REGION Network 24: Position Teaching (No 29~32)
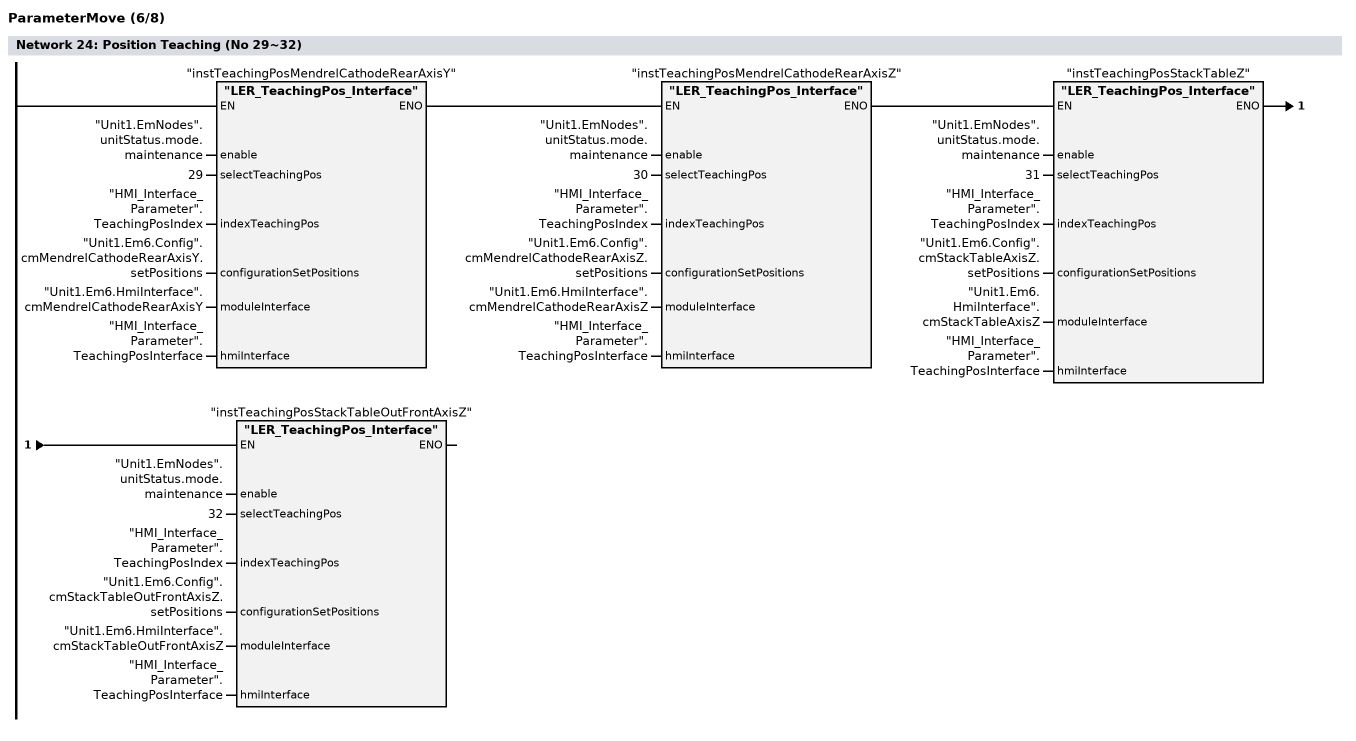
   RUNG wire#powerrail
      "instTeachingPosMendrelCathodeRearAxisY"(enable := "Unit1.EmNodes".unitStatus.mode.maintenance, selectTeachingPos := 29, indexTeachingPos := "HMI_Interface_Parameter".TeachingPosIndex, configurationSetPositions := "Unit1.Em6.Config".cmMendrelCathodeRearAxisY.setPositions, moduleInterface := "Unit1.Em6.HmiInterface".cmMendrelCathodeRearAxisY, hmiInterface := "HMI_Interface_Parameter".TeachingPosInterface)
      "instTeachingPosMendrelCathodeRearAxisZ"(enable := "Unit1.EmNodes".unitStatus.mode.maintenance, selectTeachingPos := 30, indexTeachingPos := "HMI_Interface_Parameter".TeachingPosIndex, configurationSetPositions := "Unit1.Em6.Config".cmMendrelCathodeRearAxisZ.setPositions, moduleInterface := "Unit1.Em6.HmiInterface".cmMendrelCathodeRearAxisZ, hmiInterface := "HMI_Interface_Parameter".TeachingPosInterface)
      "instTeachingPosStackTableZ"(enable := "Unit1.EmNodes".unitStatus.mode.maintenance, selectTeachingPos := 31, indexTeachingPos := "HMI_Interface_Parameter".TeachingPosIndex, configurationSetPositions := "Unit1.Em6.Config".cmStackTableAxisZ.setPositions, moduleInterface := "Unit1.Em6.HmiInterface".cmStackTableAxisZ, hmiInterface := "HMI_Interface_Parameter".TeachingPosInterface)
      "instTeachingPosStackTableOutFrontAxisZ"(enable := "Unit1.EmNodes".unitStatus.mode.maintenance, selectTeachingPos := 32, indexTeachingPos := "HMI_Interface_Parameter".TeachingPosIndex, configurationSetPositions := "Unit1.Em6.Config".cmStackTableOutFrontAxisZ.setPositions, moduleInterface := "Unit1.Em6.HmiInterface".cmStackTableOutFrontAxisZ, hmiInterface := "HMI_Interface_Parameter".TeachingPosInterface)
   END_RUNG
   // the same network as SCL:
   "instTeachingPosMendrelCathodeRearAxisY"(enable := "Unit1.EmNodes".unitStatus.mode.maintenance,   // "LER_TeachingPos_Interface"
                           selectTeachingPos := 29,
                           indexTeachingPos := "HMI_Interface_Parameter".TeachingPosIndex,
                           configurationSetPositions := "Unit1.Em6.Config".cmMendrelCathodeRearAxisY.setPositions,
                           moduleInterface := "Unit1.Em6.HmiInterface".cmMendrelCathodeRearAxisY,
                           hmiInterface := "HMI_Interface_Parameter".TeachingPosInterface,
                           ENO => #_w1);
   "instTeachingPosMendrelCathodeRearAxisZ"(EN := #_w1,   // "LER_TeachingPos_Interface"
                           enable := "Unit1.EmNodes".unitStatus.mode.maintenance,
                           selectTeachingPos := 30,
                           indexTeachingPos := "HMI_Interface_Parameter".TeachingPosIndex,
                           configurationSetPositions := "Unit1.Em6.Config".cmMendrelCathodeRearAxisZ.setPositions,
                           moduleInterface := "Unit1.Em6.HmiInterface".cmMendrelCathodeRearAxisZ,
                           hmiInterface := "HMI_Interface_Parameter".TeachingPosInterface,
                           ENO => #_w2);
   "instTeachingPosStackTableZ"(EN := #_w2,   // "LER_TeachingPos_Interface"
                           enable := "Unit1.EmNodes".unitStatus.mode.maintenance,
                           selectTeachingPos := 31,
                           indexTeachingPos := "HMI_Interface_Parameter".TeachingPosIndex,
                           configurationSetPositions := "Unit1.Em6.Config".cmStackTableAxisZ.setPositions,
                           moduleInterface := "Unit1.Em6.HmiInterface".cmStackTableAxisZ,
                           hmiInterface := "HMI_Interface_Parameter".TeachingPosInterface,
                           ENO => #_w3);
   IF #_w3 THEN
       "instTeachingPosStackTableOutFrontAxisZ"(enable := "Unit1.EmNodes".unitStatus.mode.maintenance,   // "LER_TeachingPos_Interface"
                               selectTeachingPos := 32,
                               indexTeachingPos := "HMI_Interface_Parameter".TeachingPosIndex,
                               configurationSetPositions := "Unit1.Em6.Config".cmStackTableOutFrontAxisZ.setPositions,
                               moduleInterface := "Unit1.Em6.HmiInterface".cmStackTableOutFrontAxisZ,
                               hmiInterface := "HMI_Interface_Parameter".TeachingPosInterface);
   END_IF;
END_REGION

REGION Network 25: Position Teaching (No 33~36)
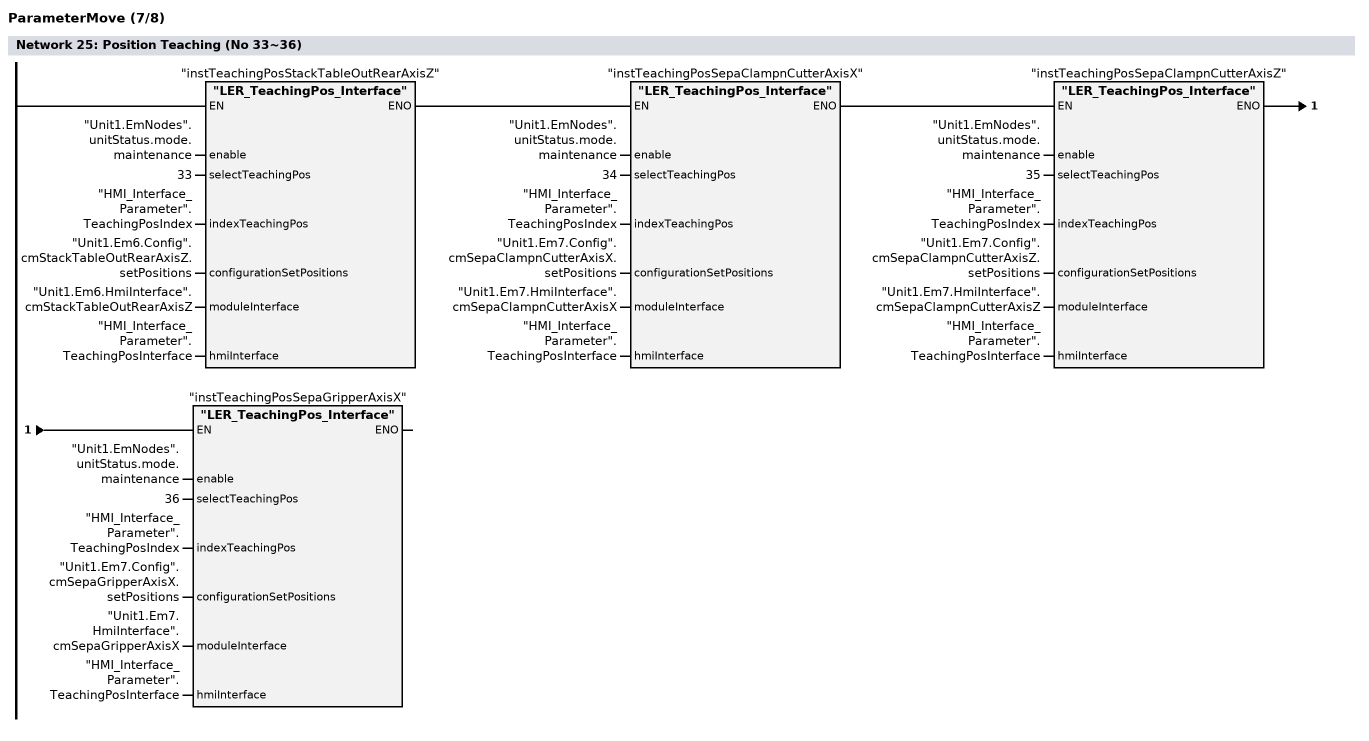
   RUNG wire#powerrail
      "instTeachingPosStackTableOutRearAxisZ"(enable := "Unit1.EmNodes".unitStatus.mode.maintenance, selectTeachingPos := 33, indexTeachingPos := "HMI_Interface_Parameter".TeachingPosIndex, configurationSetPositions := "Unit1.Em6.Config".cmStackTableOutRearAxisZ.setPositions, moduleInterface := "Unit1.Em6.HmiInterface".cmStackTableOutRearAxisZ, hmiInterface := "HMI_Interface_Parameter".TeachingPosInterface)
      "instTeachingPosSepaClampnCutterAxisX"(enable := "Unit1.EmNodes".unitStatus.mode.maintenance, selectTeachingPos := 34, indexTeachingPos := "HMI_Interface_Parameter".TeachingPosIndex, configurationSetPositions := "Unit1.Em7.Config".cmSepaClampnCutterAxisX.setPositions, moduleInterface := "Unit1.Em7.HmiInterface".cmSepaClampnCutterAxisX, hmiInterface := "HMI_Interface_Parameter".TeachingPosInterface)
      "instTeachingPosSepaClampnCutterAxisZ"(enable := "Unit1.EmNodes".unitStatus.mode.maintenance, selectTeachingPos := 35, indexTeachingPos := "HMI_Interface_Parameter".TeachingPosIndex, configurationSetPositions := "Unit1.Em7.Config".cmSepaClampnCutterAxisZ.setPositions, moduleInterface := "Unit1.Em7.HmiInterface".cmSepaClampnCutterAxisZ, hmiInterface := "HMI_Interface_Parameter".TeachingPosInterface)
      "instTeachingPosSepaGripperAxisX"(enable := "Unit1.EmNodes".unitStatus.mode.maintenance, selectTeachingPos := 36, indexTeachingPos := "HMI_Interface_Parameter".TeachingPosIndex, configurationSetPositions := "Unit1.Em7.Config".cmSepaGripperAxisX.setPositions, moduleInterface := "Unit1.Em7.HmiInterface".cmSepaGripperAxisX, hmiInterface := "HMI_Interface_Parameter".TeachingPosInterface)
   END_RUNG
   // the same network as SCL:
   "instTeachingPosStackTableOutRearAxisZ"(enable := "Unit1.EmNodes".unitStatus.mode.maintenance,   // "LER_TeachingPos_Interface"
                           selectTeachingPos := 33,
                           indexTeachingPos := "HMI_Interface_Parameter".TeachingPosIndex,
                           configurationSetPositions := "Unit1.Em6.Config".cmStackTableOutRearAxisZ.setPositions,
                           moduleInterface := "Unit1.Em6.HmiInterface".cmStackTableOutRearAxisZ,
                           hmiInterface := "HMI_Interface_Parameter".TeachingPosInterface,
                           ENO => #_w1);
   "instTeachingPosSepaClampnCutterAxisX"(EN := #_w1,   // "LER_TeachingPos_Interface"
                           enable := "Unit1.EmNodes".unitStatus.mode.maintenance,
                           selectTeachingPos := 34,
                           indexTeachingPos := "HMI_Interface_Parameter".TeachingPosIndex,
                           configurationSetPositions := "Unit1.Em7.Config".cmSepaClampnCutterAxisX.setPositions,
                           moduleInterface := "Unit1.Em7.HmiInterface".cmSepaClampnCutterAxisX,
                           hmiInterface := "HMI_Interface_Parameter".TeachingPosInterface,
                           ENO => #_w2);
   "instTeachingPosSepaClampnCutterAxisZ"(EN := #_w2,   // "LER_TeachingPos_Interface"
                           enable := "Unit1.EmNodes".unitStatus.mode.maintenance,
                           selectTeachingPos := 35,
                           indexTeachingPos := "HMI_Interface_Parameter".TeachingPosIndex,
                           configurationSetPositions := "Unit1.Em7.Config".cmSepaClampnCutterAxisZ.setPositions,
                           moduleInterface := "Unit1.Em7.HmiInterface".cmSepaClampnCutterAxisZ,
                           hmiInterface := "HMI_Interface_Parameter".TeachingPosInterface,
                           ENO => #_w3);
   IF #_w3 THEN
       "instTeachingPosSepaGripperAxisX"(enable := "Unit1.EmNodes".unitStatus.mode.maintenance,   // "LER_TeachingPos_Interface"
                               selectTeachingPos := 36,
                               indexTeachingPos := "HMI_Interface_Parameter".TeachingPosIndex,
                               configurationSetPositions := "Unit1.Em7.Config".cmSepaGripperAxisX.setPositions,
                               moduleInterface := "Unit1.Em7.HmiInterface".cmSepaGripperAxisX,
                               hmiInterface := "HMI_Interface_Parameter".TeachingPosInterface);
   END_IF;
END_REGION

REGION Network 26: Position Teaching (No 37~40)
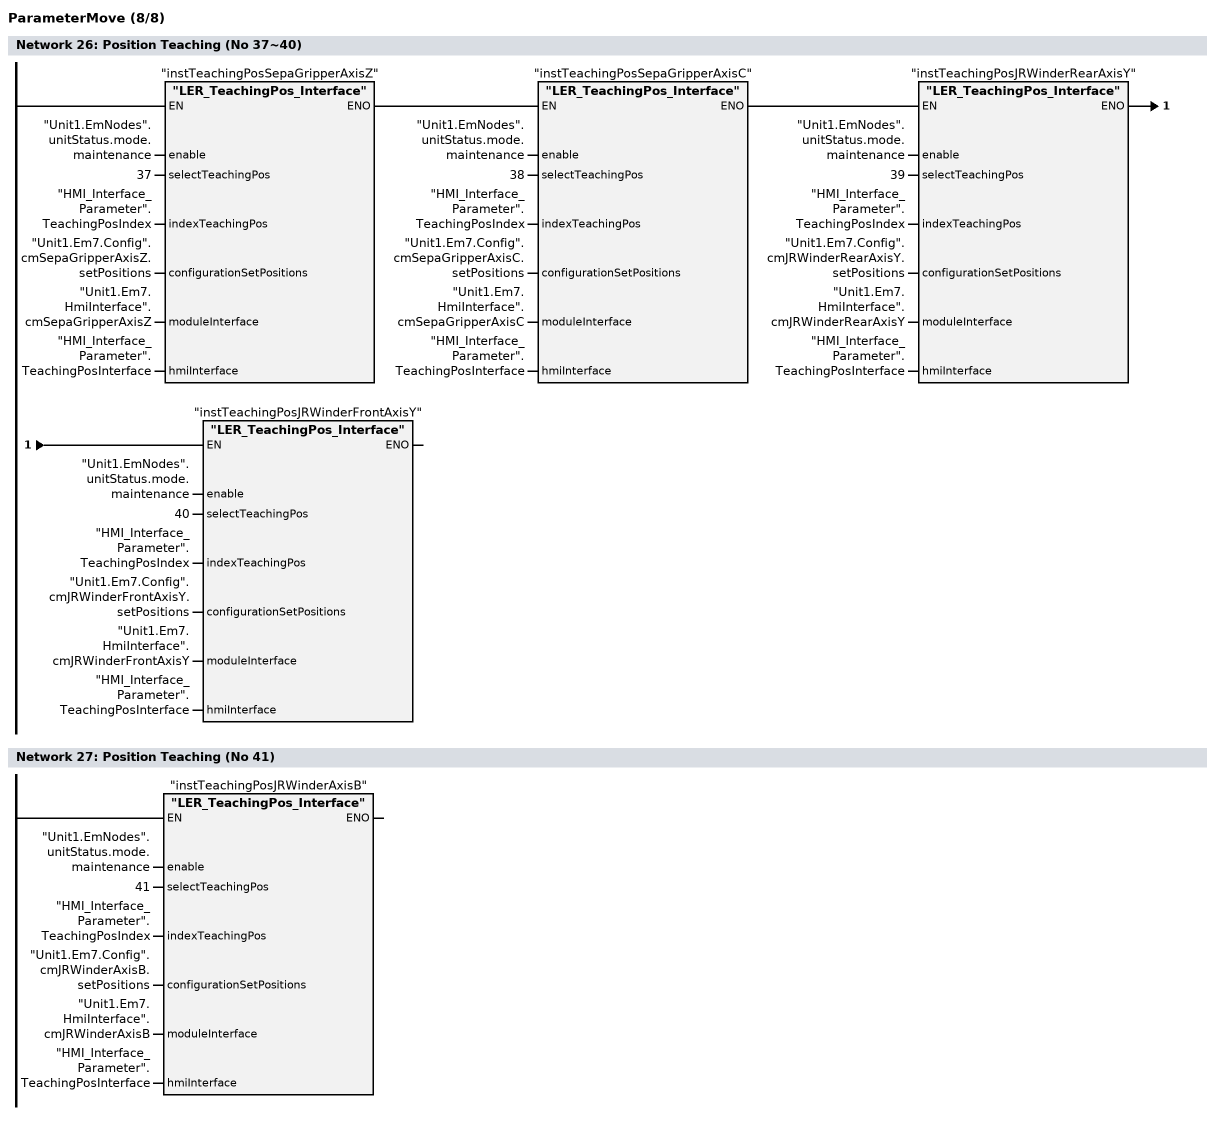
   RUNG wire#powerrail
      "instTeachingPosSepaGripperAxisZ"(enable := "Unit1.EmNodes".unitStatus.mode.maintenance, selectTeachingPos := 37, indexTeachingPos := "HMI_Interface_Parameter".TeachingPosIndex, configurationSetPositions := "Unit1.Em7.Config".cmSepaGripperAxisZ.setPositions, moduleInterface := "Unit1.Em7.HmiInterface".cmSepaGripperAxisZ, hmiInterface := "HMI_Interface_Parameter".TeachingPosInterface)
      "instTeachingPosSepaGripperAxisC"(enable := "Unit1.EmNodes".unitStatus.mode.maintenance, selectTeachingPos := 38, indexTeachingPos := "HMI_Interface_Parameter".TeachingPosIndex, configurationSetPositions := "Unit1.Em7.Config".cmSepaGripperAxisC.setPositions, moduleInterface := "Unit1.Em7.HmiInterface".cmSepaGripperAxisC, hmiInterface := "HMI_Interface_Parameter".TeachingPosInterface)
      "instTeachingPosJRWinderRearAxisY"(enable := "Unit1.EmNodes".unitStatus.mode.maintenance, selectTeachingPos := 39, indexTeachingPos := "HMI_Interface_Parameter".TeachingPosIndex, configurationSetPositions := "Unit1.Em7.Config".cmJRWinderRearAxisY.setPositions, moduleInterface := "Unit1.Em7.HmiInterface".cmJRWinderRearAxisY, hmiInterface := "HMI_Interface_Parameter".TeachingPosInterface)
      "instTeachingPosJRWinderFrontAxisY"(enable := "Unit1.EmNodes".unitStatus.mode.maintenance, selectTeachingPos := 40, indexTeachingPos := "HMI_Interface_Parameter".TeachingPosIndex, configurationSetPositions := "Unit1.Em7.Config".cmJRWinderFrontAxisY.setPositions, moduleInterface := "Unit1.Em7.HmiInterface".cmJRWinderFrontAxisY, hmiInterface := "HMI_Interface_Parameter".TeachingPosInterface)
   END_RUNG
   // the same network as SCL:
   "instTeachingPosSepaGripperAxisZ"(enable := "Unit1.EmNodes".unitStatus.mode.maintenance,   // "LER_TeachingPos_Interface"
                           selectTeachingPos := 37,
                           indexTeachingPos := "HMI_Interface_Parameter".TeachingPosIndex,
                           configurationSetPositions := "Unit1.Em7.Config".cmSepaGripperAxisZ.setPositions,
                           moduleInterface := "Unit1.Em7.HmiInterface".cmSepaGripperAxisZ,
                           hmiInterface := "HMI_Interface_Parameter".TeachingPosInterface,
                           ENO => #_w1);
   "instTeachingPosSepaGripperAxisC"(EN := #_w1,   // "LER_TeachingPos_Interface"
                           enable := "Unit1.EmNodes".unitStatus.mode.maintenance,
                           selectTeachingPos := 38,
                           indexTeachingPos := "HMI_Interface_Parameter".TeachingPosIndex,
                           configurationSetPositions := "Unit1.Em7.Config".cmSepaGripperAxisC.setPositions,
                           moduleInterface := "Unit1.Em7.HmiInterface".cmSepaGripperAxisC,
                           hmiInterface := "HMI_Interface_Parameter".TeachingPosInterface,
                           ENO => #_w2);
   "instTeachingPosJRWinderRearAxisY"(EN := #_w2,   // "LER_TeachingPos_Interface"
                           enable := "Unit1.EmNodes".unitStatus.mode.maintenance,
                           selectTeachingPos := 39,
                           indexTeachingPos := "HMI_Interface_Parameter".TeachingPosIndex,
                           configurationSetPositions := "Unit1.Em7.Config".cmJRWinderRearAxisY.setPositions,
                           moduleInterface := "Unit1.Em7.HmiInterface".cmJRWinderRearAxisY,
                           hmiInterface := "HMI_Interface_Parameter".TeachingPosInterface,
                           ENO => #_w3);
   IF #_w3 THEN
       "instTeachingPosJRWinderFrontAxisY"(enable := "Unit1.EmNodes".unitStatus.mode.maintenance,   // "LER_TeachingPos_Interface"
                               selectTeachingPos := 40,
                               indexTeachingPos := "HMI_Interface_Parameter".TeachingPosIndex,
                               configurationSetPositions := "Unit1.Em7.Config".cmJRWinderFrontAxisY.setPositions,
                               moduleInterface := "Unit1.Em7.HmiInterface".cmJRWinderFrontAxisY,
                               hmiInterface := "HMI_Interface_Parameter".TeachingPosInterface);
   END_IF;
END_REGION

REGION Network 27: Position Teaching (No 41)
   RUNG wire#powerrail
      "instTeachingPosJRWinderAxisB"(enable := "Unit1.EmNodes".unitStatus.mode.maintenance, selectTeachingPos := 41, indexTeachingPos := "HMI_Interface_Parameter".TeachingPosIndex, configurationSetPositions := "Unit1.Em7.Config".cmJRWinderAxisB.setPositions, moduleInterface := "Unit1.Em7.HmiInterface".cmJRWinderAxisB, hmiInterface := "HMI_Interface_Parameter".TeachingPosInterface)
   END_RUNG
   // the same network as SCL:
   "instTeachingPosJRWinderAxisB"(enable := "Unit1.EmNodes".unitStatus.mode.maintenance,   // "LER_TeachingPos_Interface"
                           selectTeachingPos := 41,
                           indexTeachingPos := "HMI_Interface_Parameter".TeachingPosIndex,
                           configurationSetPositions := "Unit1.Em7.Config".cmJRWinderAxisB.setPositions,
                           moduleInterface := "Unit1.Em7.HmiInterface".cmJRWinderAxisB,
                           hmiInterface := "HMI_Interface_Parameter".TeachingPosInterface);
END_REGION
END_FUNCTION
